PROGRAM CONTROLLER
VAR
	/// Freigabe Regler
	bReAktiv: BOOL := FALSE;
	/// Freigabe AWU Regler
	bAwuAktiv: BOOL := TRUE;
	/// Logger
	bLoggerRunning: BOOL := FALSE;
	fbLogger: Logger_RET;
	bFilterAktiv: BOOL;
	xy_RST_Transformation_dynamisch_0: xy_RST_Transformation_dynamisch;
	rW_x: REAL;
	rW_y: REAL;
	rX_x: REAL;
	rX_y: REAL;
	rY_x: REAL;
	rY_y: REAL;
	rY_R: REAL;
	rY_S: REAL;
	rY_T: REAL;
	bEnable_Limitierung_rY_RST: BOOL := TRUE;
	rUL_rY_RST: REAL := 150;
	rLL_rY_RST: REAL := 50;
	rE_x: REAL;
	rX_y_1: REAL;
	rX_x_1: REAL;
	
	fbFilter_X_y: PT2 := (fK := 1.0, fT1 := 0.05, fT2 := 0.05);
	fbFilter_X_x: PT2 := (fK := 1.0, fT1 := 0.05, fT2 := 0.05);
	fbSignalgeno_W_y: Signalgenerator := (eTyp := eSignalform.OFFSET, fOffset := 25.0, fAmplitude := 10.0, fFrequenz := 0.25);
	fbSignalgeno_W_x: Signalgenerator := (eTyp := eSignalform.OFFSET, fOffset := 25.0, fAmplitude := 10.0, fFrequenz := 0.25);
	fbSignalgeno_Y_x: Signalgenerator := (eTyp := eSignalform.OFFSET, fOffset := 0.0, fAmplitude := 10.0, fFrequenz := 0.25);
	fbSignalgeno_Y_y: Signalgenerator := (eTyp := eSignalform.OFFSET, fOffset := 0.0, fAmplitude := 10.0, fFrequenz := 0.25);
	fbRegler_x: Regler := (eTyp := eReglertyp.PI, fKr := 2.0, fTn := 0.2, fTv := 0.1, fTvz := 0.05, fYlim_min := 0.0, fYlim_max := 100.0, bEnable_AWU := TRUE);
	fbRegler_y: Regler := (eTyp := eReglertyp.PI, fKr := 2.0, fTn := 0.2, fTv := 0.1, fTvz := 0.05, fYlim_min := 0.0, fYlim_max := 100.0, bEnable_AWU := TRUE);
	rE_y: REAL;
	rAxisOffset: REAL := 100;
	// Zusätzlicher Filter auf Stellgrösse RST
	y_r_filter: PT1 := (fK := 1, fT := 0.05);
	y_s_filter: PT1 := (fK := 1, fT := 0.05);
	y_t_filter: PT1 := (fK := 1, fT := 0.05);
	ry_rst_filter: REAL := 0.05;  // Filterzeitkonstante PT1

END_VAR
VAR // added by the converter: edge detectors and wires of the graphical bodies
    _w1, _w2, _w3, _w4, _w7 : ANY;
    _w5, _w6, _w8, _w9 : REAL;
END_VAR

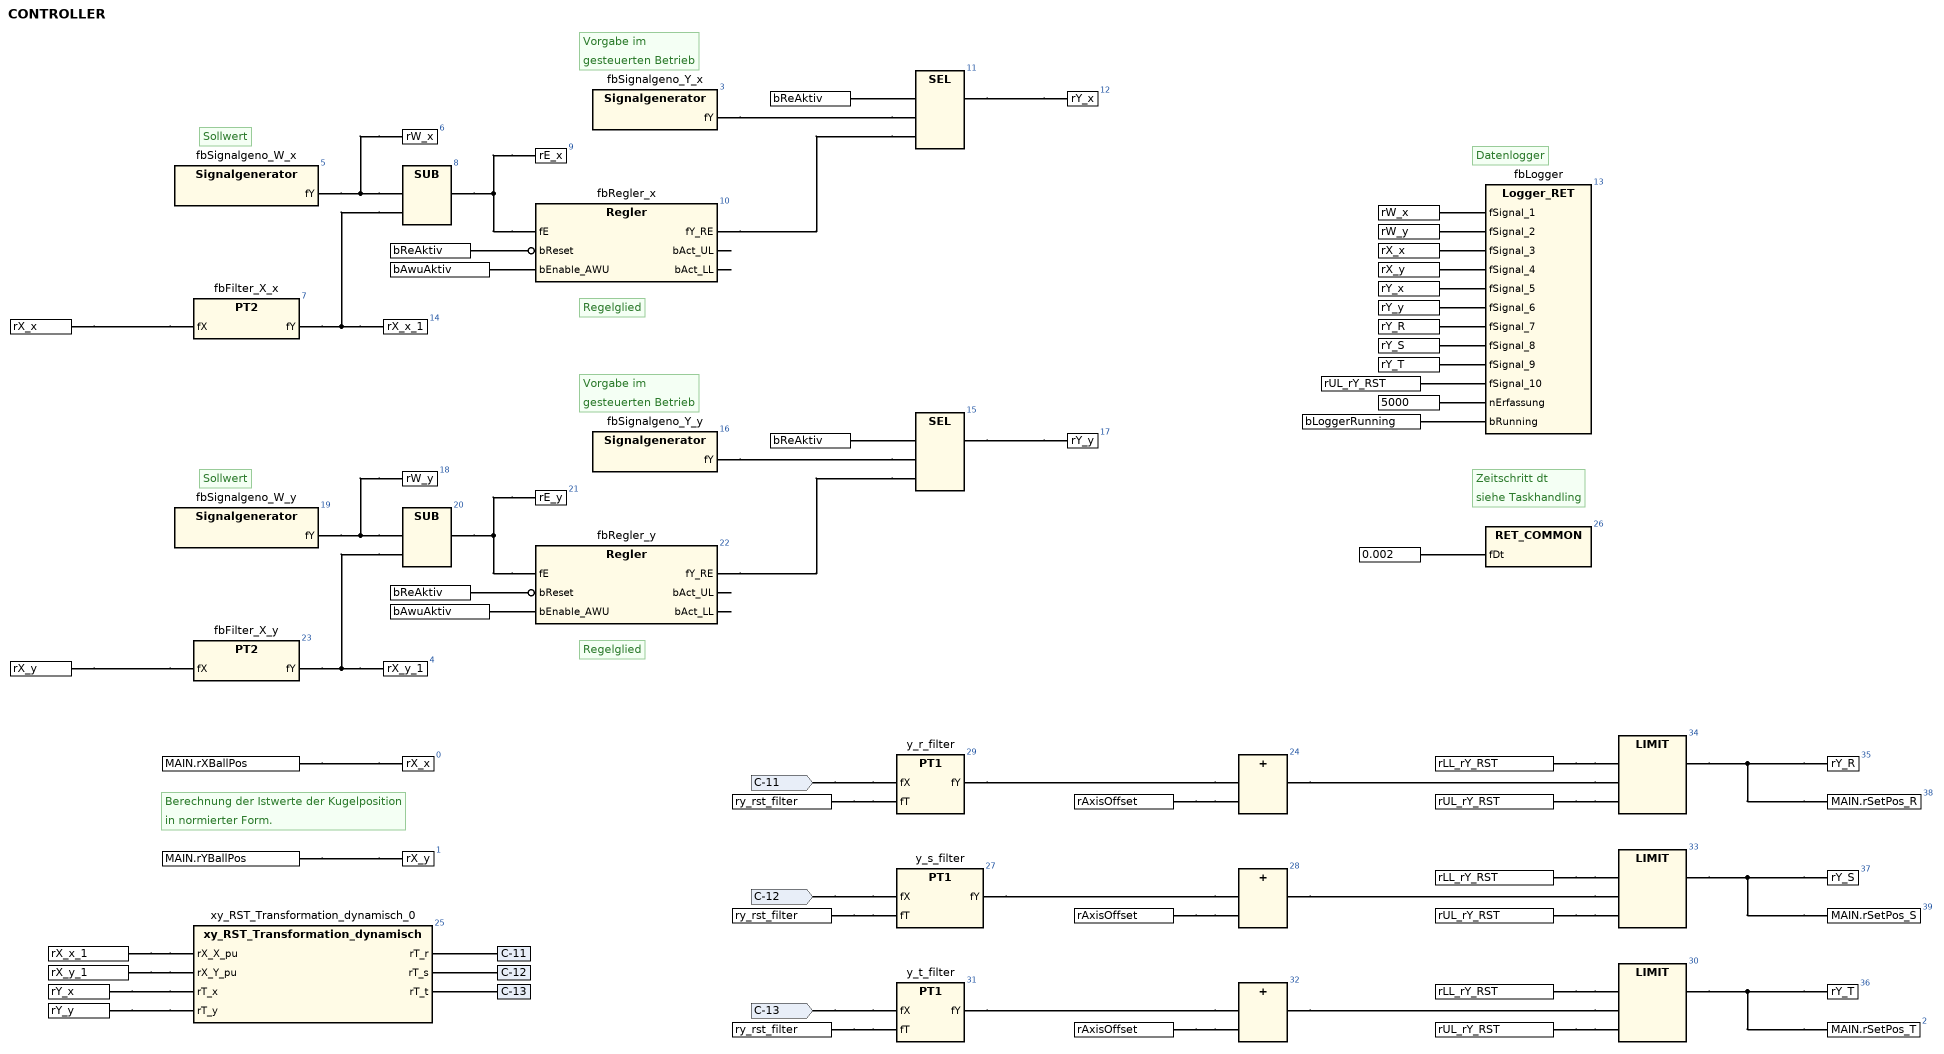
rX_x := MAIN.rXBallPos;
rX_y := MAIN.rYBallPos;
MAIN.rSetPos_T := _w1;
// Vorgabe im
// gesteuerten Betrieb
fbSignalgeno_Y_x(); // Signalgenerator
// Regelglied
rX_y_1 := fbFilter_X_y.fY;
// Sollwert
fbSignalgeno_W_x(); // Signalgenerator
rW_x := fbSignalgeno_W_x.fY;
fbFilter_X_x(fX := rX_x); // PT2
_w2 := fbSignalgeno_W_x.fY - fbFilter_X_x.fY;
rE_x := _w2;
fbRegler_x(fE := _w2, bReset := NOT bReAktiv, bEnable_AWU := bAwuAktiv); // Regler
rY_x := SEL(bReAktiv, fbSignalgeno_Y_x.fY, fbRegler_x.fY_RE);
// Datenlogger
fbLogger(
    fSignal_1 := rW_x,
    fSignal_2 := rW_y,
    fSignal_3 := rX_x,
    fSignal_4 := rX_y,
    fSignal_5 := rY_x,
    fSignal_6 := rY_y,
    fSignal_7 := rY_R,
    fSignal_8 := rY_S,
    fSignal_9 := rY_T,
    fSignal_10 := rUL_rY_RST,
    nErfassung := 5000,
    bRunning := bLoggerRunning); // Logger_RET
rX_x_1 := fbFilter_X_x.fY;
_w3 := SEL(bReAktiv, fbSignalgeno_Y_y.fY, fbRegler_y.fY_RE);
// Regelglied
// Vorgabe im
// gesteuerten Betrieb
fbSignalgeno_Y_y(); // Signalgenerator
rY_y := _w3;
rW_y := fbSignalgeno_W_y.fY;
// Sollwert
fbSignalgeno_W_y(); // Signalgenerator
_w4 := fbSignalgeno_W_y.fY - fbFilter_X_y.fY;
rE_y := _w4;
fbRegler_y(fE := _w4, bReset := NOT bReAktiv, bEnable_AWU := bAwuAktiv); // Regler
fbFilter_X_y(fX := rX_y); // PT2
_w5 := y_r_filter.fY + rAxisOffset;
// Berechnung der Istwerte der Kugelposition
// in normierter Form.
xy_RST_Transformation_dynamisch_0(rX_X_pu := rX_x_1, rX_Y_pu := rX_y_1, rT_x := rY_x, rT_y := rY_y); // xy_RST_Transformation_dynamisch
// Zeitschritt dt
// siehe Taskhandling
RET_COMMON(fDt := 0.002);
y_s_filter(fX := xy_RST_Transformation_dynamisch_0.rT_s, fT := ry_rst_filter); // PT1
_w6 := y_s_filter.fY + rAxisOffset;
y_r_filter(fX := xy_RST_Transformation_dynamisch_0.rT_r, fT := ry_rst_filter); // PT1
_w1 := LIMIT(rLL_rY_RST, _w7, rUL_rY_RST);
y_t_filter(fX := xy_RST_Transformation_dynamisch_0.rT_t, fT := ry_rst_filter); // PT1
_w7 := y_t_filter.fY + rAxisOffset;
_w8 := LIMIT(rLL_rY_RST, _w6, rUL_rY_RST);
_w9 := LIMIT(rLL_rY_RST, _w5, rUL_rY_RST);
rY_R := _w9;
rY_T := _w1;
rY_S := _w8;
MAIN.rSetPos_R := _w9;
MAIN.rSetPos_S := _w8;

END_PROGRAM

(* stored: Version 1.1.0.1, ProductVersion 3.1.4024.12
   POU CONTROLLER: Id {05086a3c-6de2-4cac-94c0-2be0236d90d4}, SpecialFunc None *)
